{attribute addProperty BoxType "EK1960-0000-0019"}
{attribute addProperty Id "FSoE_CommandUSINT811FSOUT_Module_1_Module_FaultBIT10.1251FSOUT_Module_2_Module_FaultBIT10.1251FSOUT_Module_3_Module_FaultBIT10.1251FSOUT_Module_4_Module_FaultBIT10.1251FSOUT_Module_5_Module_FaultBIT10.1251FSOUT_Module_6_Module_FaultBIT10.1251FSIN_Module_1_Channel_1_InputBIT10.1251FSIN_Module_1_Channel_2_InputBIT10.1252FSIN_Module_1_Module_FaultBIT10.1251FSIN_Module_2_Channel_1_InputBIT10.1251FSIN_Module_2_Channel_2_InputBIT10.1252FSIN_Module_2_Module_FaultBIT10.1251FSIN_Module_3_Channel_1_InputBIT10.1251FSIN_Module_3_Channel_2_InputBIT10.1252FSIN_Module_3_Module_FaultBIT10.1251FSoE_CRC_000UINT1623FSIN_Module_4_Channel_1_InputBIT10.1251FSIN_Module_4_Channel_2_InputBIT10.1252FSIN_Module_4_Module_FaultBIT10.1251FSIN_Module_5_Channel_1_InputBIT10.1251FSIN_Module_5_Channel_2_InputBIT10.1252FSIN_Module_5_Module_FaultBIT10.1251FSIN_Module_6_Channel_1_InputBIT10.1251FSIN_Module_6_Channel_2_InputBIT10.1252FSIN_Module_6_Module_FaultBIT10.1251FSIN_Module_7_Channel_1_InputBIT10.1251FSIN_Module_7_Channel_2_InputBIT10.1252FSIN_Module_7_Module_FaultBIT10.1251FSIN_Module_8_Channel_1_InputBIT10.1251FSIN_Module_8_Channel_2_InputBIT10.1252FSIN_Module_8_Module_FaultBIT10.1251FSIN_Module_9_Channel_1_InputBIT10.1251FSoE_CRC_001UINT1624FSIN_Module_9_Channel_2_InputBIT10.1252FSIN_Module_9_Module_Fault_1BIT10.1251FSIN_Module_9_Module_Fault_2BIT10.1252FSIN_Module_10_Channel_1_InputBIT10.1251FSIN_Module_10_Channel_2_InputBIT10.1252FSIN_Module_10_Module_Fault_1BIT10.1251FSIN_Module_10_Module_Fault_2BIT10.1252FSoE_CRC_002UINT1625FSoE_Connection_IDUINT1622"}
{attribute addProperty CRC "4092419179"}
{attribute addProperty SizeInBites "120"}
{attribute addProperty SizeInBytes "15"}
TYPE FSOE_F3ED5C6B :
STRUCT
	{attribute addProperty Name "FSoE_Command"}
	FSoE_Command : USINT;
	{attribute addProperty Name "FSOUT_Module_1_Module_Fault"}
	FSOUT_Module_1_Module_Fault : BIT;
	{attribute addProperty Name "FSOUT_Module_2_Module_Fault"}
	FSOUT_Module_2_Module_Fault : BIT;
	{attribute addProperty Name "FSOUT_Module_3_Module_Fault"}
	FSOUT_Module_3_Module_Fault : BIT;
	{attribute addProperty Name "FSOUT_Module_4_Module_Fault"}
	FSOUT_Module_4_Module_Fault : BIT;
	{attribute addProperty Name "FSOUT_Module_5_Module_Fault"}
	FSOUT_Module_5_Module_Fault : BIT;
	{attribute addProperty Name "FSOUT_Module_6_Module_Fault"}
	FSOUT_Module_6_Module_Fault : BIT;
	{attribute 'hide'}
	reserve_1 : BIT;
	{attribute addProperty Name "FSIN_Module_1_Channel_1_Input"}
	FSIN_Module_1_Channel_1_Input : BIT;
	{attribute addProperty Name "FSIN_Module_1_Channel_2_Input"}
	FSIN_Module_1_Channel_2_Input : BIT;
	{attribute addProperty Name "FSIN_Module_1_Module_Fault"}
	FSIN_Module_1_Module_Fault : BIT;
	{attribute addProperty Name "FSIN_Module_2_Channel_1_Input"}
	FSIN_Module_2_Channel_1_Input : BIT;
	{attribute addProperty Name "FSIN_Module_2_Channel_2_Input"}
	FSIN_Module_2_Channel_2_Input : BIT;
	{attribute addProperty Name "FSIN_Module_2_Module_Fault"}
	FSIN_Module_2_Module_Fault : BIT;
	{attribute addProperty Name "FSIN_Module_3_Channel_1_Input"}
	FSIN_Module_3_Channel_1_Input : BIT;
	{attribute addProperty Name "FSIN_Module_3_Channel_2_Input"}
	FSIN_Module_3_Channel_2_Input : BIT;
	{attribute addProperty Name "FSIN_Module_3_Module_Fault"}
	FSIN_Module_3_Module_Fault : BIT;
	{attribute addProperty Name "FSoE_CRC_000"}
	FSoE_CRC_000 : UINT;
	{attribute addProperty Name "FSIN_Module_4_Channel_1_Input"}
	FSIN_Module_4_Channel_1_Input : BIT;
	{attribute addProperty Name "FSIN_Module_4_Channel_2_Input"}
	FSIN_Module_4_Channel_2_Input : BIT;
	{attribute addProperty Name "FSIN_Module_4_Module_Fault"}
	FSIN_Module_4_Module_Fault : BIT;
	{attribute addProperty Name "FSIN_Module_5_Channel_1_Input"}
	FSIN_Module_5_Channel_1_Input : BIT;
	{attribute addProperty Name "FSIN_Module_5_Channel_2_Input"}
	FSIN_Module_5_Channel_2_Input : BIT;
	{attribute addProperty Name "FSIN_Module_5_Module_Fault"}
	FSIN_Module_5_Module_Fault : BIT;
	{attribute addProperty Name "FSIN_Module_6_Channel_1_Input"}
	FSIN_Module_6_Channel_1_Input : BIT;
	{attribute addProperty Name "FSIN_Module_6_Channel_2_Input"}
	FSIN_Module_6_Channel_2_Input : BIT;
	{attribute addProperty Name "FSIN_Module_6_Module_Fault"}
	FSIN_Module_6_Module_Fault : BIT;
	{attribute addProperty Name "FSIN_Module_7_Channel_1_Input"}
	FSIN_Module_7_Channel_1_Input : BIT;
	{attribute addProperty Name "FSIN_Module_7_Channel_2_Input"}
	FSIN_Module_7_Channel_2_Input : BIT;
	{attribute addProperty Name "FSIN_Module_7_Module_Fault"}
	FSIN_Module_7_Module_Fault : BIT;
	{attribute addProperty Name "FSIN_Module_8_Channel_1_Input"}
	FSIN_Module_8_Channel_1_Input : BIT;
	{attribute addProperty Name "FSIN_Module_8_Channel_2_Input"}
	FSIN_Module_8_Channel_2_Input : BIT;
	{attribute addProperty Name "FSIN_Module_8_Module_Fault"}
	FSIN_Module_8_Module_Fault : BIT;
	{attribute addProperty Name "FSIN_Module_9_Channel_1_Input"}
	FSIN_Module_9_Channel_1_Input : BIT;
	{attribute addProperty Name "FSoE_CRC_001"}
	FSoE_CRC_001 : UINT;
	{attribute addProperty Name "FSIN_Module_9_Channel_2_Input"}
	FSIN_Module_9_Channel_2_Input : BIT;
	{attribute addProperty Name "FSIN_Module_9_Module_Fault_1"}
	FSIN_Module_9_Module_Fault_1 : BIT;
	{attribute addProperty Name "FSIN_Module_9_Module_Fault_2"}
	FSIN_Module_9_Module_Fault_2 : BIT;
	{attribute addProperty Name "FSIN_Module_10_Channel_1_Input"}
	FSIN_Module_10_Channel_1_Input : BIT;
	{attribute addProperty Name "FSIN_Module_10_Channel_2_Input"}
	FSIN_Module_10_Channel_2_Input : BIT;
	{attribute addProperty Name "FSIN_Module_10_Module_Fault_1"}
	FSIN_Module_10_Module_Fault_1 : BIT;
	{attribute addProperty Name "FSIN_Module_10_Module_Fault_2"}
	FSIN_Module_10_Module_Fault_2 : BIT;
	{attribute 'hide'}
	reserve_2_BIT_0 : BIT;
	{attribute 'hide'}
	reserve_2_BIT_1 : BIT;
	{attribute 'hide'}
	reserve_2_BIT_2 : BIT;
	{attribute 'hide'}
	reserve_2_BIT_3 : BIT;
	{attribute 'hide'}
	reserve_2_BIT_4 : BIT;
	{attribute 'hide'}
	reserve_2_BIT_5 : BIT;
	{attribute 'hide'}
	reserve_2_BIT_6 : BIT;
	{attribute 'hide'}
	reserve_2_BIT_7 : BIT;
	{attribute 'hide'}
	reserve_2_BIT_8 : BIT;
	{attribute addProperty Name "FSoE_CRC_002"}
	FSoE_CRC_002 : UINT;
	{attribute addProperty Name "FSoE_Connection_ID"}
	FSoE_Connection_ID : UINT;
END_STRUCT
END_TYPE

(* stored: Version 1.2.0.0, ProductVersion 3.1.4024.9
   DUT FSOE_F3ED5C6B: Id {b29d8613-bfff-4dd4-8c8a-5984ca894445} *)
